# EPICS substitutions: iocBoot/iocoh26/substitutions/fb_epid.substitutions
# $Id$

file "$(OPTICS)/opticsApp/Db/fb_epid.db"
  {
    {
        P=oh26:epid1,
	IN=oh26:epid1:sim.VAL,
	OUT=oh26:epid1:sim.D,
	MODE=PID,
	CALC=A,
	PERMIT1="oh26:epid1:on.VAL",
	PERMIT2="",
	PERMIT3="",
	PERMIT4=""
    }
  }
